% RSLogix 500 project Industrial Pump Control with HOA and Safety Alarms – RSLogix 500.RSS, saved by version 8.30.00.16 %
PROJECT "UNTITLED"    % processor: Bul.1763 MicroLogix 1100 Series B %

PROGRAM FILES
  LAD 2   5 rungs
  LAD 3 "IO"  8 rungs
  LAD 4 "CTRL LOGIC"  7 rungs
  LAD 5 "ALRM LOGIC"  9 rungs
  LAD 6 "HOA"  6 rungs

DATA FILES
  O0 OUTPUT  4 elements
  I1 INPUT  6 elements
  S2 STATUS  66 elements
  B3 BINARY  2 elements
  T4 TIMER  4 elements
  C5 COUNTER  1 elements
  R6 CONTROL  1 elements
  N7 INTEGER  3 elements
  F8 FLOAT  1 elements

LADDER 2
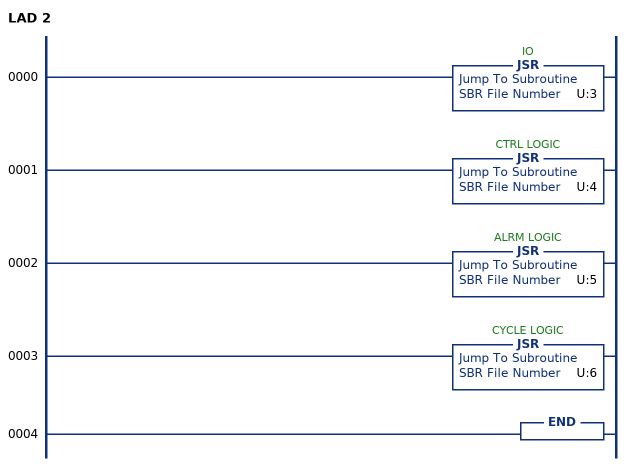
% Rung: 0 %
SOR JSR U:3 EOR
%   U:3  "IO" %
% Rung: 1 %
SOR JSR U:4 EOR
%   U:4  "CTRL LOGIC" %
% Rung: 2 %
SOR JSR U:5 EOR
%   U:5  "ALRM LOGIC" %
% Rung: 3 %
SOR JSR U:6 EOR
%   U:6  "CYCLE LOGIC" %
% Rung: 4 %
SOR END EOR

LADDER 3 "IO"
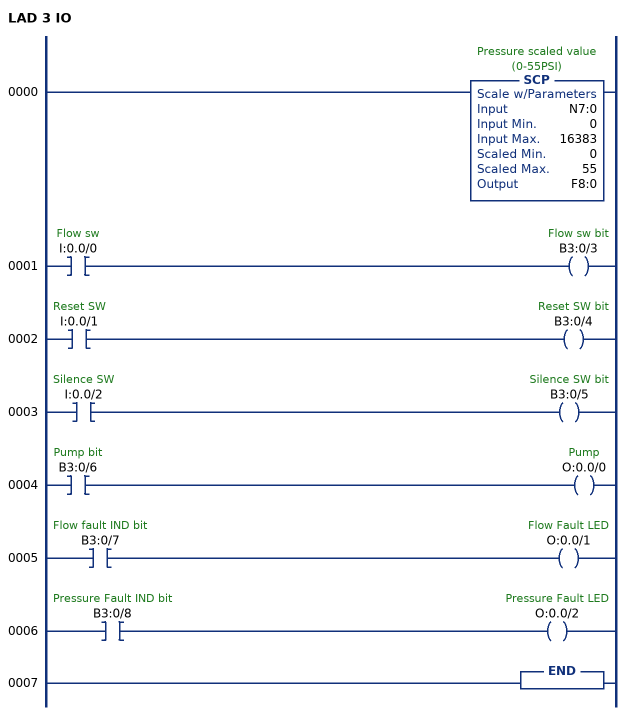
% Rung: 0 %
SOR SCP N7:0 0 16383 0 55 F8:0 EOR
%   N7:0  "Pressure Check" %
%   F8:0  "Pressure scaled value (0-55PSI)" %
% Rung: 1 %
SOR XIC I:0.0/0 OTE B3:0/3 EOR
%   I:0.0/0  "Flow sw" %
%   B3:0/3  "Flow sw bit" %
% Rung: 2 %
SOR XIC I:0.0/1 OTE B3:0/4 EOR
%   I:0.0/1  "Reset SW" %
%   B3:0/4  "Reset SW bit" %
% Rung: 3 %
SOR XIC I:0.0/2 OTE B3:0/5 EOR
%   I:0.0/2  "Silence SW" %
%   B3:0/5  "Silence SW bit" %
% Rung: 4 %
SOR XIC B3:0/6 OTE O:0.0/0 EOR
%   B3:0/6  "Pump bit" %
%   O:0.0/0  "Pump" %
% Rung: 5 %
SOR XIC B3:0/7 OTE O:0.0/1 EOR
%   B3:0/7  "Flow fault IND bit" %
%   O:0.0/1  "Flow Fault LED" %
% Rung: 6 %
SOR XIC B3:0/8 OTE O:0.0/2 EOR
%   B3:0/8  "Pressure Fault IND bit" %
%   O:0.0/2  "Pressure Fault LED" %
% Rung: 7 %
SOR END EOR

LADDER 4 "CTRL LOGIC"
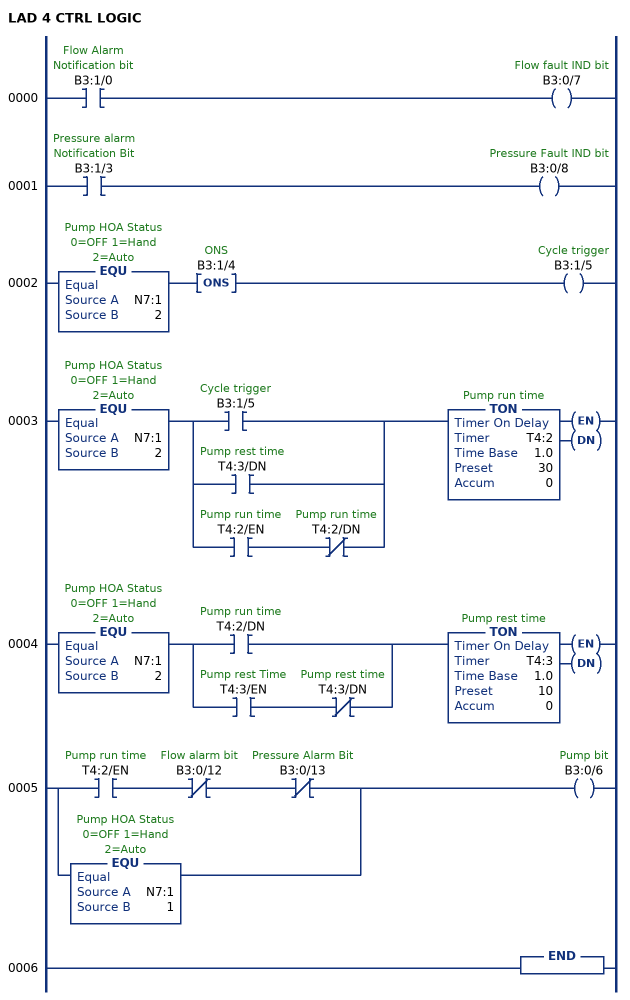
% Rung: 0 %
SOR XIC B3:1/0 OTE B3:0/7 EOR
%   B3:1/0  "Flow Alarm Notification bit" %
%   B3:0/7  "Flow fault IND bit" %
% Rung: 1 %
SOR XIC B3:1/3 OTE B3:0/8 EOR
%   B3:1/3  "Pressure alarm Notification Bit" %
%   B3:0/8  "Pressure Fault IND bit" %
% Rung: 2 %
SOR EQU N7:1 2 ONS B3:1/4 OTE B3:1/5 EOR
%   N7:1  "Pump HOA Status 0=OFF 1=Hand 2=Auto" %
%   B3:1/4  "ONS" %
%   B3:1/5  "Cycle trigger" %
% Rung: 3 %
SOR EQU N7:1 2 BST BST XIC B3:1/5 NXB XIC T4:3/DN BND NXB XIC T4:2/EN XIO T4:2/DN BND TON T4:2 1.0 30 0 EOR
%   N7:1  "Pump HOA Status 0=OFF 1=Hand 2=Auto" %
%   B3:1/5  "Cycle trigger" %
%   T4:3/DN  "Pump rest time" %
%   T4:2/EN  "Pump run time" %
%   T4:2/DN  "Pump run time" %
%   T4:2  "Pump run time" %
% Rung: 4 %
SOR EQU N7:1 2 BST XIC T4:2/DN NXB XIC T4:3/EN XIO T4:3/DN BND TON T4:3 1.0 10 0 EOR
%   N7:1  "Pump HOA Status 0=OFF 1=Hand 2=Auto" %
%   T4:2/DN  "Pump run time" %
%   T4:3/EN  "Pump rest Time" %
%   T4:3/DN  "Pump rest time" %
%   T4:3  "Pump rest time" %
% Rung: 5 %
SOR BST XIC T4:2/EN XIO B3:0/12 XIO B3:0/13 NXB EQU N7:1 1 BND OTE B3:0/6 EOR
%   T4:2/EN  "Pump run time" %
%   B3:0/12  "Flow alarm bit" %
%   B3:0/13  "Pressure Alarm Bit" %
%   N7:1  "Pump HOA Status 0=OFF 1=Hand 2=Auto" %
%   B3:0/6  "Pump bit" %
% Rung: 6 %
SOR END EOR

LADDER 5 "ALRM LOGIC"
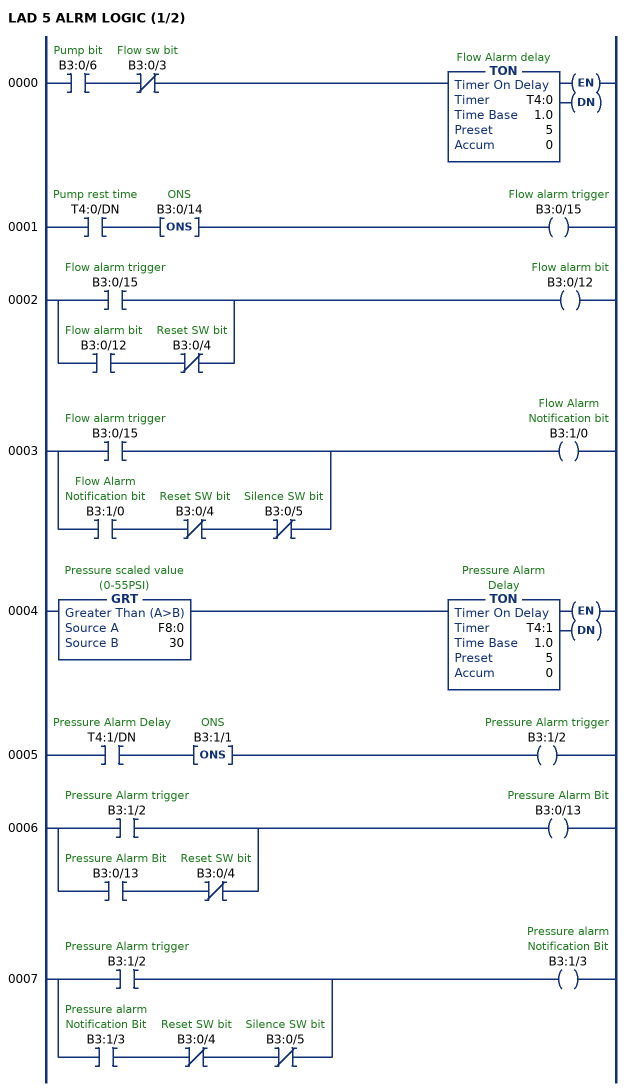
% Rung: 0 %
SOR XIC B3:0/6 XIO B3:0/3 TON T4:0 1.0 5 0 EOR
%   B3:0/6  "Pump bit" %
%   B3:0/3  "Flow sw bit" %
%   T4:0  "Flow Alarm delay" %
% Rung: 1 %
SOR XIC T4:0/DN ONS B3:0/14 OTE B3:0/15 EOR
%   T4:0/DN  "Pump rest time" %
%   B3:0/14  "ONS" %
%   B3:0/15  "Flow alarm trigger" %
% Rung: 2 %
SOR BST XIC B3:0/15 NXB XIC B3:0/12 XIO B3:0/4 BND OTE B3:0/12 EOR
%   B3:0/15  "Flow alarm trigger" %
%   B3:0/12  "Flow alarm bit" %
%   B3:0/4  "Reset SW bit" %
% Rung: 3 %
SOR BST XIC B3:0/15 NXB XIC B3:1/0 XIO B3:0/4 XIO B3:0/5 BND OTE B3:1/0 EOR
%   B3:0/15  "Flow alarm trigger" %
%   B3:1/0  "Flow Alarm Notification bit" %
%   B3:0/4  "Reset SW bit" %
%   B3:0/5  "Silence SW bit" %
% Rung: 4 %
SOR GRT F8:0 30 TON T4:1 1.0 5 0 EOR
%   F8:0  "Pressure scaled value (0-55PSI)" %
%   T4:1  "Pressure Alarm Delay" %
% Rung: 5 %
SOR XIC T4:1/DN ONS B3:1/1 OTE B3:1/2 EOR
%   T4:1  "Pressure Alarm Delay" %
%   B3:1/1  "ONS" %
%   B3:1/2  "Pressure Alarm trigger" %
% Rung: 6 %
SOR BST XIC B3:1/2 NXB XIC B3:0/13 XIO B3:0/4 BND OTE B3:0/13 EOR
%   B3:1/2  "Pressure Alarm trigger" %
%   B3:0/13  "Pressure Alarm Bit" %
%   B3:0/4  "Reset SW bit" %
% Rung: 7 %
SOR BST XIC B3:1/2 NXB XIC B3:1/3 XIO B3:0/4 XIO B3:0/5 BND OTE B3:1/3 EOR
%   B3:1/2  "Pressure Alarm trigger" %
%   B3:1/3  "Pressure alarm Notification Bit" %
%   B3:0/4  "Reset SW bit" %
%   B3:0/5  "Silence SW bit" %

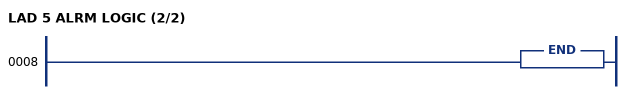
% Rung: 8 %
SOR END EOR

LADDER 6 "HOA"
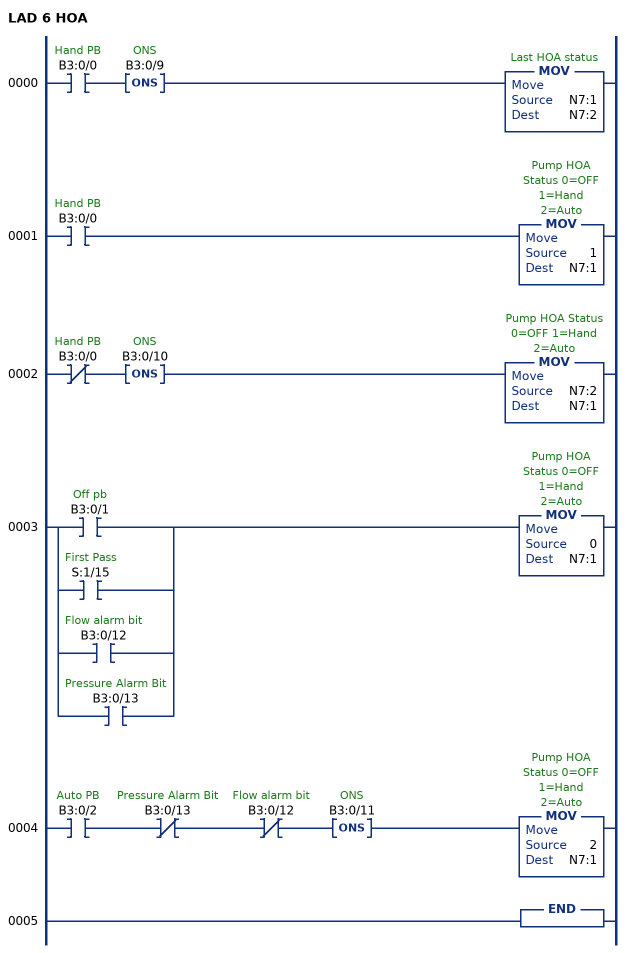
% Rung: 0 %
SOR XIC B3:0/0 ONS B3:0/9 MOV N7:1 N7:2 EOR
%   B3:0/0  "Hand PB" %
%   B3:0/9  "ONS" %
%   N7:1  "Pump HOA Status 0=OFF 1=Hand 2=Auto" %
%   N7:2  "Last HOA status" %
% Rung: 1 %
SOR XIC B3:0/0 MOV 1 N7:1 EOR
%   B3:0/0  "Hand PB" %
%   N7:1  "Pump HOA Status 0=OFF 1=Hand 2=Auto" %
% Rung: 2 %
SOR XIO B3:0/0 ONS B3:0/10 MOV N7:2 N7:1 EOR
%   B3:0/0  "Hand PB" %
%   B3:0/10  "ONS" %
%   N7:2  "Last HOA status" %
%   N7:1  "Pump HOA Status 0=OFF 1=Hand 2=Auto" %
% Rung: 3 %
SOR BST XIC B3:0/1 NXB XIC S:1/15 NXB XIC B3:0/12 NXB XIC B3:0/13 BND MOV 0 N7:1 EOR
%   B3:0/1  "Off pb" %
%   S:1/15  "First Pass" %
%   B3:0/12  "Flow alarm bit" %
%   B3:0/13  "Pressure Alarm Bit" %
%   N7:1  "Pump HOA Status 0=OFF 1=Hand 2=Auto" %
% Rung: 4 %
SOR XIC B3:0/2 XIO B3:0/13 XIO B3:0/12 ONS B3:0/11 MOV 2 N7:1 EOR
%   B3:0/2  "Auto PB" %
%   B3:0/13  "Pressure Alarm Bit" %
%   B3:0/12  "Flow alarm bit" %
%   B3:0/11  "ONS" %
%   N7:1  "Pump HOA Status 0=OFF 1=Hand 2=Auto" %
% Rung: 5 %
SOR END EOR

OTHER DOCUMENTED ADDRESSES
  U:7  "OUTPUT LOGIC"

DATA TABLE (non-zero values as saved)
DATA T4
% .PRE .ACC %
% T4:0 % 5 0
% T4:1 % 5 0
% T4:2 % 30 0
% T4:3 % 10 0
